FUNCTION_BLOCK EL2002
VAR
	{attribute addProperty Name "WcState"}
	_wcState : WcStateBase;
	{attribute addProperty Name "Info data"}
	_infoData : InfoDataBase;
	_io : EL2xx2_Data;
END_VAR

PROPERTY IO : REFERENCE TO EL2xx2_Data
GET
IO REF= _io;
END_GET
END_PROPERTY

PROPERTY WcState : REFERENCE TO WcStateBase
GET
WcState REF= _wcState;
END_GET
END_PROPERTY

END_FUNCTION_BLOCK

(* stored: Version 1.1.0.1, ProductVersion 3.1.4024.9
   POU EL2002: Id {5efaaa2e-772e-0b60-0dab-527280492888}, SpecialFunc None
   Property IO: Id {2f183b06-5e54-0699-0842-91b67082eeb6}
   Get Get: Id {40e39f84-d812-062a-35c4-fe3f67693ffd}
   Property WcState: Id {33550a72-377e-0512-14cf-5f18b7f59ee9}
   Get Get: Id {dd51b7ef-fdac-0170-271d-5670cad39f93} *)
